// TwinCAT 3 PLC project WP_Controller
// ProgramVersion: 3.1.4024.0
// libraries:
//   Tc2_MC2, * (Beckhoff Automation GmbH)
//   Tc2_ModbusRTU, * (Beckhoff Automation GmbH)
//   Tc2_Standard, * (Beckhoff Automation GmbH)
//   Tc2_System, * (Beckhoff Automation GmbH)
//   Tc2_Utilities, * (Beckhoff Automation GmbH)
//   Tc3_Module, * (Beckhoff Automation GmbH)
//   Tc3_Vision, * (Beckhoff Automation GmbH)
// project tree:
//   GVLs/ GVL.TcGVL
//   / PlcTask.TcTTO, VisionTask.TcTTO (not stored)
//   POUs/ FB_ClockPulse.TcPOU, FB_EnableAxes.TcPOU, FB_StrASCConversion.TcPOU (not stored), F_Scale.TcPOU, MAIN.TcPOU, PRG_LoadcellScaling.TcPOU, PRG_PLCModbusRTU.TcPOU (not stored), PRG_MotorDrive.TcPOU, PRG_PneumaticValves.TcPOU, PRG_PowerMeasurement.TcPOU, PRG_SafetyLightCurtain.TcPOU, PRG_Thermocouple.TcPOU, PRG_VfdModbusRtu.TcPOU, VISION.TcPOU (not stored)
// real-time tasks:
//   TASK PlcTask: cycle T#10ms, priority 20, ADS port 350
//   TASK VisionTask: cycle T#10ms, priority 21, ADS port 351
//   TASK VnTask ImgAcq (FileSource1): cycle T#10ms, priority 5, ADS port 352
//   TASK VnTask ImgAcq (Camera1): cycle T#1ms, priority 6, ADS port 353
//   TASK VnTask ADS (Camera1): cycle T#10ms, priority 7, ADS port 354
// motion (NC):
//   TASK NC-Task 1 SAF: cycle T#2ms, priority 4, ADS port 501
//   TASK NC-Task 1 SVB: cycle T#10ms, priority 8, ADS port 511
//   AXIS Axis 1 (id 1)
//     OtherSettings: AllowMotionCmdToSlave=true
//     encoder EncType=1
//     drive DrvType=5
//       Analog: TorqueSetpointScale=10, ScaleFactorActTorque=0.1
//       TimeComp: TaskDelayCycles=1
//     controller CtrType=1
//       CtrPara: PriorControlFactor=1
//         Observer: BandWidth=20
//   AXIS Axis 2 (id 2)
//     OtherSettings: AllowMotionCmdToSlave=true
//     encoder EncType=4
//       EncPara: MaxCount=#x0000ffff
//         Inc: RefSoftSyncMask=#x0000ffff
//     drive DrvType=24
//       Analog: TorqueSetpointScale=10, ScaleFactorActTorque=0.1
//       TimeComp: TaskDelayCycles=1
//     controller CtrType=1
//       CtrPara: PriorControlFactor=1
//         Observer: BandWidth=20
// I/O:
//   DEVICE Device 5 (EtherCAT), AmsNetId 169.254.69.6.6.1
//     Term 1 (EK1100) [EK1100 EtherCAT Coupler (2A E-Bus)]
//       Term 2 (EL7031) [EL7031 1Ch. Stepper motor output stage (24V, 1.5A)]
//       Term 3 (EL2596) [EL2596 1-channel LED strobe control terminal 24V/3A]
//       Term 4 (EL9011) [EL9011 End Terminal]
//   DEVICE Device 1 (RT-Ethernet Adapter)
// variable links:
//   NC-Task 1 SAF/Axes/Axis 2 <-> Device 5 (EtherCAT)/Term 1 (EK1100)/Term 2 (EL7031)
//     Drive/Inputs/In/nState1 @bit 3 <-> STM Status/Status/Error
//     Drive/Inputs/In/nState1 @bit 5 <-> STM Status/Status/Moving negative
//     Drive/Inputs/In/nState1 @bit 4 <-> STM Status/Status/Moving positive
//     Drive/Inputs/In/nState1 @bit 1 <-> STM Status/Status/Ready
//     Drive/Inputs/In/nState1 <-> STM Status/Status/Ready to enable
//     Drive/Inputs/In/nState1 @bit 6 <-> STM Status/Status/Torque reduced
//     Drive/Inputs/In/nState1 @bit 2 <-> STM Status/Status/Warning
//     Drive/Inputs/In/nState2 @bit 3 <-> STM Status/Status/Digital input 1
//     Drive/Inputs/In/nState2 @bit 4 <-> STM Status/Status/Digital input 2
//     Drive/Inputs/In/nState2 @bit 5 <-> STM Status/Status/Sync error
//     Drive/Inputs/In/nState2 @bit 7 <-> STM Status/Status/TxPDO Toggle
//     Drive/Inputs/In/nState4 @bit 1 <-> WcState/InputToggle
//     Drive/Inputs/In/nState4 <-> WcState/WcState
//     Drive/Outputs/Out/nCtrl1 <-> STM Control/Control/Enable
//     Drive/Outputs/Out/nCtrl1 @bit 2 <-> STM Control/Control/Reduce torque
//     Drive/Outputs/Out/nCtrl1 @bit 1 <-> STM Control/Control/Reset
//     Drive/Outputs/Out/nDataOut2[0] <-> STM Velocity/Velocity
//     Enc/Inputs/In/nDataIn1[0] <-> ENC Status compact/Counter value
//     Enc/Inputs/In/nDataIn2[0] <-> ENC Status compact/Latch value
//     Enc/Inputs/In/nState1 @bit 4 <-> ENC Status compact/Status/Counter overflow
//     Enc/Inputs/In/nState1 @bit 3 <-> ENC Status compact/Status/Counter underflow
//     Enc/Inputs/In/nState1 @bit 1 <-> ENC Status compact/Status/Latch extern valid
//     Enc/Inputs/In/nState1 @bit 2 <-> ENC Status compact/Status/Set counter done
//     Enc/Inputs/In/nState2 @bit 4 <-> ENC Status compact/Status/Status of extern latch
//     Enc/Inputs/In/nState2 @bit 5 <-> ENC Status compact/Status/Sync error
//     Enc/Inputs/In/nState2 @bit 7 <-> ENC Status compact/Status/TxPDO Toggle
//     Enc/Inputs/In/nState4 @bit 1 <-> WcState/InputToggle
//     Enc/Inputs/In/nState4 <-> WcState/WcState
//     Enc/Outputs/Out/nCtrl1 @bit 3 <-> ENC Control compact/Control/Enable latch extern on negative edge
//     Enc/Outputs/Out/nCtrl1 @bit 1 <-> ENC Control compact/Control/Enable latch extern on positive edge
//     Enc/Outputs/Out/nCtrl1 @bit 2 <-> ENC Control compact/Control/Set counter
//     Enc/Outputs/Out/nDataOut1[0] <-> ENC Control compact/Set counter value
//   WP_Controller/WP_Controller Instance <-> NC-Task 1 SAF/Axes/Axis 1
//     PlcTask Inputs/GVL.stAxis1.NcToPlc <-> Outputs/ToPlc
//     PlcTask Outputs/GVL.stAxis1.PlcToNc <-> Inputs/FromPlc

CONFIGURATION WP_Controller
    RESOURCE PLC ON TwinCAT3
        TASK PlcTask(INTERVAL := T#10ms, PRIORITY := 20);
        PROGRAM MAIN WITH PlcTask : MAIN;
    END_RESOURCE
END_CONFIGURATION

// ---- GVLs/GVL.TcGVL
{attribute 'qualified_only'}
VAR_GLOBAL
	//Thermocouple
	nTemp AT %I*: INT;
	
	//Power measurement
	// RMS Current
	fIL1 AT %I*: REAL;
	fIL2 AT %I*: REAL;
	fIL3 AT %I*: REAL;
	
	//RMS Voltage
	fUL1 AT %I*: REAL;
	fUL2 AT %I*: REAL;
	fUL3 AT %I*: REAL;
	
	//Active Power
	fActivePower AT %I* : REAL;
	
	// Phase angle
	fcosphi1 AT %I*: REAL;
	fcosphi2 AT %I*: REAL;
	fcosphi3 AT %I*: REAL;
	
	// Frequency
	fFrequency AT %I*: REAL;
	
	//Motor drive
	stAxis1: AXIS_REF;
	bButtonFw AT %I*: BOOL; //Self reset
	bButtonBw AT %I*: BOOL; //Self reset
	bButtonHalt AT %I*: BOOL; //Self reset
	bButtonAuto AT %I*: BOOL; //Latch
	
	//VFD Modbus RTU
	bEnable AT %I*: BOOL; //Self reset
	bDisable AT %I*: BOOL; //Self reset
	
	// Bit 0 and Bit 1 declaration
	bModbusCoilBit0 : BOOL;
	bModbusCoilBit1 : BOOL;
	
	// Virtual toggle buttons for write values using MODBUS RTU
	bExecuteWriteCoils: BOOL:=TRUE;
	bExecuteWriteRegs0: BOOL;
	//bExecuteWriteRegs1: BOOL;

	// Input STRING from HMI, MAXIMUM 20 characters
	sInputFromHMI: STRING(20);		

	//Constant value for testing, used for EL2596
	bLedEnable AT %Q*:BOOL:=TRUE;
	bLedOutput AT %Q*:BOOL:=TRUE;
	bOutputCurrent AT %Q*: UINT:=300;
	
	// Constant value for EL2809 controlling strobe
	bLedEnableEL2xxx AT %Q*:BOOL:=TRUE; 
	
	// Loadcell scaling variables
	uLoadCellRawValue AT %I*: DINT;
	uLoadCellScaledValue: REAL;
	
	// Output signal variables for sneumatic valves 
	bValve1 AT %Q*:BOOL;
	bValve2 AT %Q*:BOOL;
	bValve3 AT %Q*:BOOL;
	bValve4 AT %Q*:BOOL;
	bValve5 AT %Q*:BOOL;
	bValve6 AT %Q*:BOOL;
	bVirtualToggleButton1:BOOL;
	bVirtualToggleButton2:BOOL;
	bVirtualToggleButton3:BOOL;
	bVirtualToggleButton4:BOOL;
	bVirtualToggleButton5:BOOL;
	bVirtualToggleButton6:BOOL;
	
	// TwinSAFE declaration
	bSafeRun AT %Q*:BOOL;
	bSafeAck AT %Q*:BOOL;
	bSafeFBErr AT %I*: BOOL;
	bSafeCommErr AT %I*: BOOL;
	bSafeRedLedOutput AT %Q*:BOOL; // safety output signal for EL2809 
	bSafeRedLedInput AT %I*:BOOL; // safety red led reception signal for ouput signal imported from EL6910
	bSafeRestartSignal AT %Q*: BOOL; //restart signal for safeESTop FB
	bSafeRestartSignalInput AT %I*: BOOL; //restart signal
	
	
END_VAR

// ---- POUs/MAIN.TcPOU
PROGRAM MAIN
VAR
END_VAR

PRG_Thermocouple();
PRG_PowerMeasurement();
PRG_MotorDrive();
PRG_PneumaticValves();
PRG_PLCModbusRTU();
PRG_LoadcellScaling();
PRG_SafetyLightCurtain();

END_PROGRAM

// ---- POUs/PRG_Thermocouple.TcPOU
PROGRAM PRG_Thermocouple
VAR
	fTemp: REAL;
END_VAR

fTemp := GVL.nTemp;

END_PROGRAM

// ---- POUs/PRG_PowerMeasurement.TcPOU
PROGRAM PRG_PowerMeasurement
VAR
	fActivePowerAbs: REAL;
	fIL1Abs: REAL;
	fIL2Abs: REAL;
	fIL3Abs: REAL;
END_VAR

fActivePowerAbs := ABS(GVL.fActivePower);
fIL1Abs := ABS(GVL.fIL1);
fIL2Abs := ABS(GVL.fIL2);
fIL3Abs := ABS(GVL.fIL3);

END_PROGRAM

// ---- POUs/PRG_MotorDrive.TcPOU
PROGRAM PRG_MotorDrive
VAR
	fbEnableAxes: FB_EnableAxes;
	fbHalt1: MC_Halt;
	fbMoveVelocityFw: MC_MoveVelocity;
	fbMoveVelocityBw: MC_MoveVelocity;
	fbTON1: TON;
	fbRTrigMoveFw: R_TRIG;
	fbRTrigMoveBw: R_TRIG;
	fbRTrigHalt: R_TRIG;
	nAutoState: INT;
END_VAR

fbEnableAxes.bEnableAxes := TRUE;
fbRTrigMoveFW(CLK:=GVL.bButtonFw, Q=>);
fbRTrigMoveBW(CLK:=GVL.bButtonBw, Q=>);
fbRTrigHalt(CLK:=GVL.bButtonHalt, Q=>);

IF fbRTrigMoveFw.Q THEN
	fbHalt1.Execute := FALSE;
	fbMoveVelocityBw.Execute := FALSE;
	fbMoveVelocityFw.Execute := TRUE;
END_IF

IF fbRTrigMoveBw.Q THEN
	fbHalt1.Execute := FALSE;
	fbMoveVelocityFw.Execute := FALSE;
	fbMoveVelocityBw.Execute := TRUE;
END_IF

IF fbRTrigHalt.Q THEN
	fbHalt1.Execute := TRUE;
	fbMoveVelocityFw.Execute := FALSE;
	fbMoveVelocityBw.Execute := FALSE;
END_IF

IF GVL.bButtonAuto THEN
	CASE nAutoState OF
		0: //Initialize auto motion
			fbHalt1.Execute := FALSE;
			fbMoveVelocityFw.Execute := FALSE;
			fbMoveVelocityBw.Execute := FALSE;
			nAutoState := 1;
		1: //Move forward
			fbTON1(IN:=TRUE, PT:=T#4S, Q=>, ET=>);
			fbMoveVelocityFw.Execute := TRUE;
			IF fbTON1.Q THEN
				fbTON1(IN:=FALSE);
				nAutoState := 2;	
			END_IF
		2: //Halt
			fbTON1(IN:=TRUE, PT:=T#2S, Q=>, ET=>);
			fbMoveVelocityFw.Execute := FALSE;
			fbHalt1.Execute := TRUE;
			IF fbTON1.Q THEN
				fbTON1(IN:=FALSE);
				nAutoState := 3;	
			END_IF
		3: //Move backward
			fbTON1(IN:=TRUE, PT:=T#4S, Q=>, ET=>);
			fbHalt1.Execute := FALSE;
			fbMoveVelocityBw.Execute := TRUE;
			IF fbTON1.Q THEN
				fbTON1(IN:=FALSE);
				nAutoState := 4;	
			END_IF
		4: //Halt again
			fbTON1(IN:=TRUE, PT:=T#2S, Q=>, ET=>);
			fbMoveVelocityBw.Execute := FALSE;
			fbHalt1.Execute := TRUE;
			IF fbTON1.Q THEN
				fbTON1(IN:=FALSE);
				nAutoState := 0;	
			END_IF
	END_CASE
END_IF

A_EnableAxes();
A_MoveVelocityFw();
A_MoveVelocityBw();
A_Halt();

ACTION A_EnableAxes:
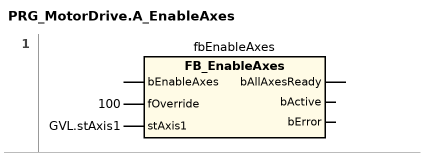
// NETWORK 1
fbEnableAxes(fOverride := 100, stAxis1 := GVL.stAxis1); // FB_EnableAxes
END_ACTION

ACTION A_Halt:
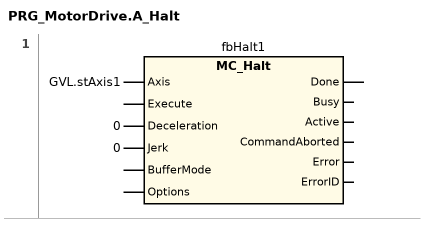
// NETWORK 1
fbHalt1(Axis := GVL.stAxis1, Deceleration := 0, Jerk := 0); // MC_Halt
END_ACTION

ACTION A_MoveVelocityBw:
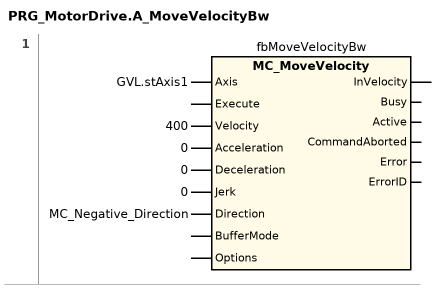
// NETWORK 1
fbMoveVelocityBw(
    Axis := GVL.stAxis1,
    Velocity := 400,
    Acceleration := 0,
    Deceleration := 0,
    Jerk := 0,
    Direction := MC_Negative_Direction); // MC_MoveVelocity
END_ACTION

ACTION A_MoveVelocityFw:
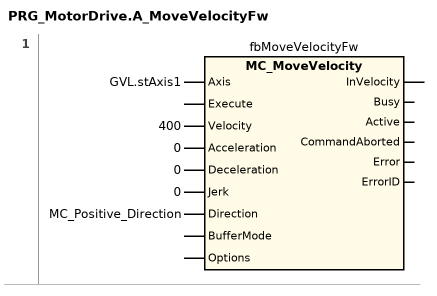
// NETWORK 1
fbMoveVelocityFw(
    Axis := GVL.stAxis1,
    Velocity := 400,
    Acceleration := 0,
    Deceleration := 0,
    Jerk := 0,
    Direction := MC_Positive_Direction); // MC_MoveVelocity
END_ACTION

END_PROGRAM

// ---- POUs/FB_EnableAxes.TcPOU
FUNCTION_BLOCK FB_EnableAxes
VAR_INPUT
	bEnableAxes			: BOOL;
	fOverride			: LREAL;
END_VAR
VAR_OUTPUT
	bAllAxesReady		: BOOL;
	bActive				: BOOL;
	bError				: BOOL;
END_VAR
VAR_IN_OUT
	stAxis1				: AXIS_REF;
END_VAR
VAR
	fbPower1			:MC_Power;
END_VAR

fbPower1(
	Enable:=bEnableAxes, 
	Enable_Positive:=bEnableAxes, 
	Enable_Negative:=bEnableAxes, 
	Override:=fOverride, 
	BufferMode:= , 
	Axis:=stAxis1, 
	Status=> , 
	Busy=> , 
	Active=> , 
	Error=> , 
	ErrorID=> );

IF fbPower1.Active THEN
	bActive := TRUE;
	IF fbPower1.Error THEN
		bError := TRUE;
	ELSE 
		bAllAxesReady := fbPower1.Status;
		bError := FALSE;
	END_IF
ELSE
	bActive := FALSE;
END_IF

END_FUNCTION_BLOCK

// ---- POUs/PRG_PneumaticValves.TcPOU
PROGRAM PRG_PneumaticValves
VAR
END_VAR

// Valve 1
IF GVL.bVirtualToggleButton1 THEN
	GVL.bValve1:=TRUE;
ELSE
	GVL.bValve1:=FALSE;
END_IF

// Valve2
IF GVL.bVirtualToggleButton2 THEN
	GVL.bValve2:=TRUE;
ELSE
	GVL.bValve2:=FALSE;
END_IF

// Valve 3
IF GVL.bVirtualToggleButton3 THEN
	GVL.bValve3:=TRUE;
ELSE
	GVL.bValve3:=FALSE;
END_IF


// Valve 4
IF GVL.bVirtualToggleButton4 THEN
	GVL.bValve4:=TRUE;
ELSE
	GVL.bValve4:=FALSE;
END_IF

// Valve 5
IF GVL.bVirtualToggleButton5 THEN
	GVL.bValve5:=TRUE;
ELSE
	GVL.bValve5:=FALSE;
END_IF

// Valve 6
IF GVL.bVirtualToggleButton6 THEN
	GVL.bValve6:=TRUE;
ELSE
	GVL.bValve6:=FALSE;
END_IF

END_PROGRAM

// ---- POUs/PRG_LoadcellScaling.TcPOU
PROGRAM PRG_LoadcellScaling
VAR
END_VAR

GVL.uLoadCellScaledValue := F_Scale(GVL.uLoadCellRawValue, 0.0, 1.0, -383, 1200);

END_PROGRAM

// ---- POUs/F_Scale.TcPOU
FUNCTION F_Scale : REAL
VAR_INPUT
	nAIn: DINT;
	fOutMin: REAL; // Maximum of the output value
	fOutMax: REAL; // Minimum of the output value
	nInMin: DINT; // Minimum of the input value
	nInMax: DINT; // Maximum of the input value
END_VAR
VAR
	fAIn: REAL;
	fSlope: REAL;
	fConstant: REAL;
	fInMax: REAL;
	fInMin: REAL;
END_VAR

// Binding rules
IF nAIn >= nInMax THEN
	nAIN := nInMax;
ELSIF nAIn <= nInMin THEN
	nAIn := nInMin;
END_IF

fAIn := DINT_TO_REAL(nAIn);
fInMax := DINT_TO_REAL(nInMax);
fInMin := DINT_TO_REAL(nInMin);

// y = ax + b

// Find a
fSlope := (fOutMax-fOutMin)/(fInMax-fInMin);

// Find b
fConstant := fOutMin - (fSlope * fInMin);

F_Scale := fSlope*fAin + fConstant;

END_FUNCTION

// ---- POUs/PRG_SafetyLightCurtain.TcPOU
PROGRAM PRG_SafetyLightCurtain
VAR
END_VAR

GVL.bSafeRedLedOutput := GVL.bSafeRedLedInput;
GVL.bSafeRestartSignal:=GVL.bSafeRestartSignalInput;

END_PROGRAM

// ---- POUs/FB_ClockPulse.TcPOU
FUNCTION_BLOCK FB_ClockPulse
VAR_INPUT
	bStart:BOOL;
END_VAR
VAR_OUTPUT
	bExecute: BOOL;
END_VAR
VAR
	fbTimer1, fbTimer2: TON;
END_VAR

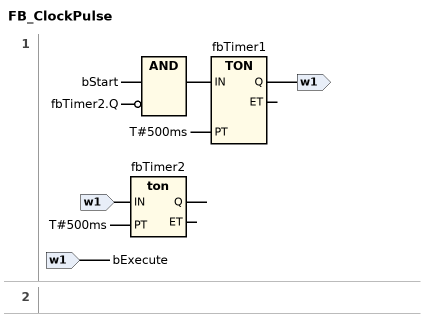
// NETWORK 1
fbTimer1(IN := bStart AND NOT fbTimer2.Q, PT := T#500ms); // TON
fbTimer2(IN := fbTimer1.Q, PT := T#500ms); // ton
bExecute := fbTimer1.Q;

// NETWORK 2

END_FUNCTION_BLOCK

// ---- POUs/PRG_VfdModbusRtu.TcPOU
PROGRAM PRG_VfdModbusRtu
VAR
	fbVfdMb: ModbusRtuMaster_KL6x22B;
	fbRTrigWrite: R_Trig;
	fbRTrigEnable: R_Trig;
	fbRTrigDisable: R_Trig;
	fbTON: TON;
	wQty: WORD := 1;
	wMbAddr: WORD;
	wCmd: WORD;
	bWrite: BOOL;
END_VAR

fbRTrigWrite(CLK:=bWrite, Q=>);
fbRTrigEnable(CLK:=GVL.bEnable, Q=>);
fbRTrigEnable(CLK:=GVL.bDisable, Q=>);

IF fbRTrigEnable.Q THEN
	bWrite := TRUE;
	fbTON(IN:= bWrite, PT:= T#500MS, Q=> , ET=> );
	wMbAddr := 416;
	wCmd := 1;
END_IF

IF fbRTrigDisable.Q THEN
	bWrite := TRUE;
	fbTON(IN:= bWrite, PT:= T#500MS, Q=> , ET=> );
	wMbAddr := 416;
	wCmd := 0;
END_IF

IF fbTON.Q THEN
	fbTON(IN:=FALSE);
	bWrite := FALSE;
END_IF

fbVfdMb.WriteRegs(
	UnitID:= 1, 
	Quantity:= wQty, 
	MBAddr:= wMbAddr, 
	cbLength:= SIZEOF(wCmd), 
	pMemoryAddr:= ADR(wCmd), 
	Execute:= fbRTrigWrite.Q, 
	Timeout:= T#1S, 
	BUSY=> , 
	Error=> , 
	ErrorId=> , 
	cbRead=> );

END_PROGRAM
